{attribute addProperty BoxType "EL3413-0000-0016"}
{attribute addProperty Id "OvervoltageBIT10.1251UndervoltageBIT10.1252OvercurrentBIT10.1253Phase_sequence_cwBIT10.1255Phase_sequence_ccwBIT10.1256Missing_zero_crossingBIT10.1257TxPDO_StateBIT10.12515TxPDO_ToggleBIT10.12516"}
{attribute addProperty CRC "982537029"}
{attribute addProperty SizeInBites "16"}
{attribute addProperty SizeInBytes "2"}
TYPE STATUS_3A905345 :
STRUCT
	{attribute addProperty Name "Overvoltage"}
	Overvoltage : BIT;
	{attribute addProperty Name "Undervoltage"}
	Undervoltage : BIT;
	{attribute addProperty Name "Overcurrent"}
	Overcurrent : BIT;
	{attribute 'hide'}
	reserve_1 : BIT;
	{attribute addProperty Name "Phase_sequence_cw"}
	Phase_sequence_cw : BIT;
	{attribute addProperty Name "Phase_sequence_ccw"}
	Phase_sequence_ccw : BIT;
	{attribute addProperty Name "Missing_zero_crossing"}
	Missing_zero_crossing : BIT;
	{attribute 'hide'}
	reserve_2_BIT_0 : BIT;
	{attribute 'hide'}
	reserve_2_BIT_1 : BIT;
	{attribute 'hide'}
	reserve_2_BIT_2 : BIT;
	{attribute 'hide'}
	reserve_2_BIT_3 : BIT;
	{attribute 'hide'}
	reserve_2_BIT_4 : BIT;
	{attribute 'hide'}
	reserve_2_BIT_5 : BIT;
	{attribute 'hide'}
	reserve_2_BIT_6 : BIT;
	{attribute addProperty Name "TxPDO_State"}
	TxPDO_State : BIT;
	{attribute addProperty Name "TxPDO_Toggle"}
	TxPDO_Toggle : BIT;
END_STRUCT
END_TYPE

(* stored: Version 1.2.0.0, ProductVersion 3.1.4024.9
   DUT STATUS_3A905345: Id {b766804c-4fbb-417c-bf61-c4ee03ecc270} *)
